// TIA Portal V18 export
FUNCTION "SS1_A4_4AO_IO_Update" : Void   // FC11040, LAD
{ S7_Optimized_Access := 'TRUE' }
VERSION : 0.1
// stored: AutoNumber false, IsIECCheckEnabled false, SetENOAutomatically false, UDAEnableTagReadback false
BEGIN

REGION Network 1: AO0
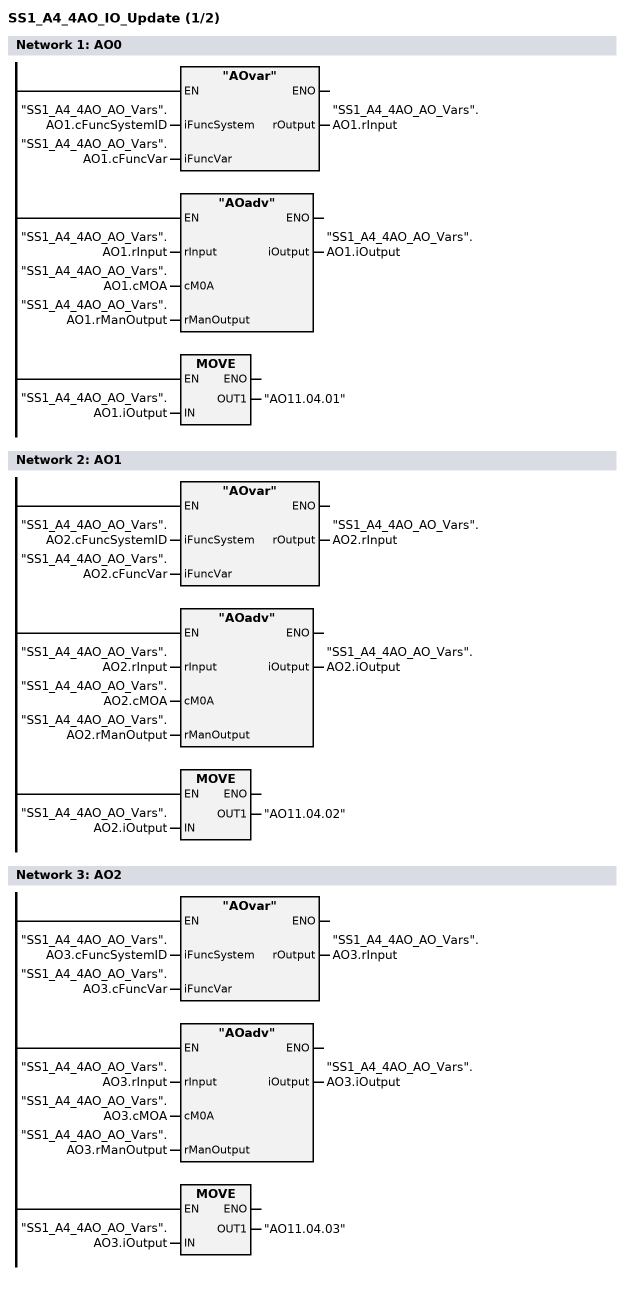
   RUNG wire#powerrail
      "AOvar"(iFuncSystem := "SS1_A4_4AO_AO_Vars".AO1.cFuncSystemID, iFuncVar := "SS1_A4_4AO_AO_Vars".AO1.cFuncVar, rOutput => "SS1_A4_4AO_AO_Vars".AO1.rInput)
   END_RUNG
   RUNG wire#powerrail
      "AOadv"(rInput := "SS1_A4_4AO_AO_Vars".AO1.rInput, cM0A := "SS1_A4_4AO_AO_Vars".AO1.cMOA, rManOutput := "SS1_A4_4AO_AO_Vars".AO1.rManOutput, iOutput => "SS1_A4_4AO_AO_Vars".AO1.iOutput)
   END_RUNG
   RUNG wire#powerrail
      Move(in := "SS1_A4_4AO_AO_Vars".AO1.iOutput, out1 => "AO11.04.01")
   END_RUNG
   // the same network as SCL:
   "AOvar"(iFuncSystem := "SS1_A4_4AO_AO_Vars".AO1.cFuncSystemID,
           iFuncVar := "SS1_A4_4AO_AO_Vars".AO1.cFuncVar,
           rOutput => "SS1_A4_4AO_AO_Vars".AO1.rInput);
   "AOadv"(rInput := "SS1_A4_4AO_AO_Vars".AO1.rInput,
           cM0A := "SS1_A4_4AO_AO_Vars".AO1.cMOA,
           rManOutput := "SS1_A4_4AO_AO_Vars".AO1.rManOutput,
           iOutput => "SS1_A4_4AO_AO_Vars".AO1.iOutput);
   "AO11.04.01" := "SS1_A4_4AO_AO_Vars".AO1.iOutput;
END_REGION

REGION Network 2: AO1
   RUNG wire#powerrail
      "AOvar"(iFuncSystem := "SS1_A4_4AO_AO_Vars".AO2.cFuncSystemID, iFuncVar := "SS1_A4_4AO_AO_Vars".AO2.cFuncVar, rOutput => "SS1_A4_4AO_AO_Vars".AO2.rInput)
   END_RUNG
   RUNG wire#powerrail
      "AOadv"(rInput := "SS1_A4_4AO_AO_Vars".AO2.rInput, cM0A := "SS1_A4_4AO_AO_Vars".AO2.cMOA, rManOutput := "SS1_A4_4AO_AO_Vars".AO2.rManOutput, iOutput => "SS1_A4_4AO_AO_Vars".AO2.iOutput)
   END_RUNG
   RUNG wire#powerrail
      Move(in := "SS1_A4_4AO_AO_Vars".AO2.iOutput, out1 => "AO11.04.02")
   END_RUNG
   // the same network as SCL:
   "AOvar"(iFuncSystem := "SS1_A4_4AO_AO_Vars".AO2.cFuncSystemID,
           iFuncVar := "SS1_A4_4AO_AO_Vars".AO2.cFuncVar,
           rOutput => "SS1_A4_4AO_AO_Vars".AO2.rInput);
   "AOadv"(rInput := "SS1_A4_4AO_AO_Vars".AO2.rInput,
           cM0A := "SS1_A4_4AO_AO_Vars".AO2.cMOA,
           rManOutput := "SS1_A4_4AO_AO_Vars".AO2.rManOutput,
           iOutput => "SS1_A4_4AO_AO_Vars".AO2.iOutput);
   "AO11.04.02" := "SS1_A4_4AO_AO_Vars".AO2.iOutput;
END_REGION

REGION Network 3: AO2
   RUNG wire#powerrail
      "AOvar"(iFuncSystem := "SS1_A4_4AO_AO_Vars".AO3.cFuncSystemID, iFuncVar := "SS1_A4_4AO_AO_Vars".AO3.cFuncVar, rOutput => "SS1_A4_4AO_AO_Vars".AO3.rInput)
   END_RUNG
   RUNG wire#powerrail
      "AOadv"(rInput := "SS1_A4_4AO_AO_Vars".AO3.rInput, cM0A := "SS1_A4_4AO_AO_Vars".AO3.cMOA, rManOutput := "SS1_A4_4AO_AO_Vars".AO3.rManOutput, iOutput => "SS1_A4_4AO_AO_Vars".AO3.iOutput)
   END_RUNG
   RUNG wire#powerrail
      Move(in := "SS1_A4_4AO_AO_Vars".AO3.iOutput, out1 => "AO11.04.03")
   END_RUNG
   // the same network as SCL:
   "AOvar"(iFuncSystem := "SS1_A4_4AO_AO_Vars".AO3.cFuncSystemID,
           iFuncVar := "SS1_A4_4AO_AO_Vars".AO3.cFuncVar,
           rOutput => "SS1_A4_4AO_AO_Vars".AO3.rInput);
   "AOadv"(rInput := "SS1_A4_4AO_AO_Vars".AO3.rInput,
           cM0A := "SS1_A4_4AO_AO_Vars".AO3.cMOA,
           rManOutput := "SS1_A4_4AO_AO_Vars".AO3.rManOutput,
           iOutput => "SS1_A4_4AO_AO_Vars".AO3.iOutput);
   "AO11.04.03" := "SS1_A4_4AO_AO_Vars".AO3.iOutput;
END_REGION

REGION Network 4: AO3
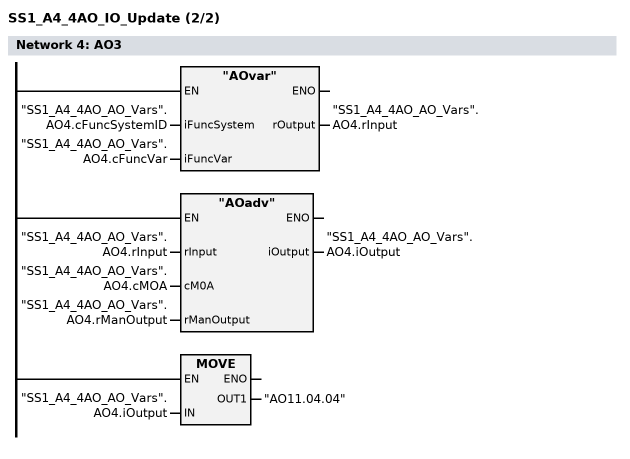
   RUNG wire#powerrail
      "AOvar"(iFuncSystem := "SS1_A4_4AO_AO_Vars".AO4.cFuncSystemID, iFuncVar := "SS1_A4_4AO_AO_Vars".AO4.cFuncVar, rOutput => "SS1_A4_4AO_AO_Vars".AO4.rInput)
   END_RUNG
   RUNG wire#powerrail
      "AOadv"(rInput := "SS1_A4_4AO_AO_Vars".AO4.rInput, cM0A := "SS1_A4_4AO_AO_Vars".AO4.cMOA, rManOutput := "SS1_A4_4AO_AO_Vars".AO4.rManOutput, iOutput => "SS1_A4_4AO_AO_Vars".AO4.iOutput)
   END_RUNG
   RUNG wire#powerrail
      Move(in := "SS1_A4_4AO_AO_Vars".AO4.iOutput, out1 => "AO11.04.04")
   END_RUNG
   // the same network as SCL:
   "AOvar"(iFuncSystem := "SS1_A4_4AO_AO_Vars".AO4.cFuncSystemID,
           iFuncVar := "SS1_A4_4AO_AO_Vars".AO4.cFuncVar,
           rOutput => "SS1_A4_4AO_AO_Vars".AO4.rInput);
   "AOadv"(rInput := "SS1_A4_4AO_AO_Vars".AO4.rInput,
           cM0A := "SS1_A4_4AO_AO_Vars".AO4.cMOA,
           rManOutput := "SS1_A4_4AO_AO_Vars".AO4.rManOutput,
           iOutput => "SS1_A4_4AO_AO_Vars".AO4.iOutput);
   "AO11.04.04" := "SS1_A4_4AO_AO_Vars".AO4.iOutput;
END_REGION
END_FUNCTION
